FUNCTION_BLOCK FB_Control2 EXTENDS FB_BaseControlElement IMPLEMENTS ITF_Control1, ITF_Control2_HMI_Connector
VAR
END_VAR

END_FUNCTION_BLOCK

(* stored: Version 1.1.0.1
   POU FB_Control2: Id {5a1fda2c-d90a-09fa-2335-09f6611015bb}, SpecialFunc None *)
